{attribute addProperty BoxType "EK1100-0000-0018"}
{attribute addProperty Id "Beckhoff_EP4xxxEK1122Beckhoff_EP4xxxEK1122_2529070E2032254"}
{attribute addProperty CRC "427707794"}
{attribute addProperty SizeInBites "2032"}
{attribute addProperty SizeInBytes "254"}
TYPE Beckhoff_EP4xxx_197E4D92 EXTENDS EK1100_179A0949 :
STRUCT
	{attribute addProperty Name "Beckhoff_EP4xxxEK1122"}
	Beckhoff_EP4xxxEK1122 : Beckhoff_EP4xxxEK1122_2529070E;
END_STRUCT
END_TYPE

(* stored: Version 1.2.0.0, ProductVersion 3.1.4024.9
   DUT Beckhoff_EP4xxx_197E4D92: Id {448e3264-531e-4e7c-be8c-914d31dfa0ff} *)
